FUNCTION_BLOCK _HRESULT_TestSuite EXTENDS TcUnit.FB_TestSuite
VAR
END_VAR

TestAddress();
TestClearReference();
TestClone();
TestTypeNameReturnsExpected();
TestIdentifierReturnsExpected();
TestMakeReferenceToFollowsReference();
TestMakeReferenceToUpdatesReference();
TestSize();
TestValueReturnsExpectedAfterInit();
TestValueReturnsExpectedAfterChange();
TestSerializeTypeWith();
TestSerializeWith();
TestTryDeserializeFrom();
TestTryMakeReferenceToFollowsReference();
TestTryMakeReferenceToUpdatesReference();

METHOD PUBLIC TestAddress
VAR
    _type : _HRESULT(S_OK);
    notExpected : PVOID := 0;
    actual : PVOID;
END_VAR
TEST('TestAddress');

actual := _type.Address;

AssertFalse(
    Condition := (notExpected = actual),
    Message := 'Type did not return a valid address.'
);

TEST_FINISHED();
END_METHOD

METHOD PUBLIC TestClearReference
VAR
    _type : _HRESULT(S_OK);
	target : HRESULT := S_OK;
    expected : HRESULT := S_OK;
    actual : HRESULT;
END_VAR
TEST('TestClearReference');

_type.MakeReferenceTo(target);
_type.ClearReference();
target := S_FALSE;

actual := _type.Value;

AssertEquals(
    Expected := expected,
    Actual := actual,
    Message := 'Value did not follow target change'
);

TEST_FINISHED();
END_METHOD

METHOD PUBLIC TestClone
VAR
    _type : _HRESULT(S_OK);
	clone : I_Datatype;
	isValidClone : BOOL;
	compareResult : DINT;
END_VAR
TEST('TestClone');

clone := _type.Clone();

isValidClone := clone <> 0;

IF isValidClone THEN
	compareResult := memcmp(_type.Address, clone.Address, clone.Size);
END_IF

AssertTrue(
	Condition := isValidClone,
	Message := 'Clone did not produce a clone'
);

AssertEquals_DINT(
	Expected := 0,
    Actual := compareResult,
    Message := 'Clone did not return a valid clone.'
);

clone.Dispose();

TEST_FINISHED();
END_METHOD

METHOD PUBLIC TestIdentifierReturnsExpected
VAR
    _type : _HRESULT(S_OK);
    expected : STRING := 'HRESULT';
    actual : STRING;
END_VAR
TEST('TestIdentifierReturnsExpected');

actual := _type.Identifier;

AssertEquals_STRING(
    Expected := expected,
    Actual := actual,
    Message := 'Type did not return correct iec type.'
);

TEST_FINISHED();
END_METHOD

METHOD PUBLIC TestMakeReferenceToFollowsReference
VAR
    _type : _HRESULT(S_OK);
	target : HRESULT := S_OK;
    expected : HRESULT := S_FALSE;
    actual : HRESULT;
END_VAR
TEST('TestMakeReferenceToFollowsReference');

_type.MakeReferenceTo(target);
target := S_FALSE;

actual := _type.Value;

AssertEquals(
    Expected := expected,
    Actual := actual,
    Message := 'Value did not follow target change'
);

TEST_FINISHED();
END_METHOD

METHOD PUBLIC TestMakeReferenceToUpdatesReference
VAR
    _type : _HRESULT(S_OK);
	target : HRESULT := S_OK;
    expected : HRESULT := S_FALSE;
    actual : HRESULT;
END_VAR
TEST('TestMakeReferenceToUpdatesReference');

_type.MakeReferenceTo(target);
_type.Value := S_FALSE;

actual := target;

AssertEquals(
    Expected := expected,
    Actual := actual,
    Message := 'Value did not update target'
);

TEST_FINISHED();
END_METHOD

METHOD PUBLIC TestSerializeTypeWith
VAR
    _type : _HRESULT(S_OK);
    serializer : JsonSerializer;
    expected : STRING(500) := '{"typeName":"ALIAS","identifier":"HRESULT","baseDatatype":{"typeName":"DINT","minValue":-2147483648,"maxValue":2147483647,"isSigned":true,"isFloat":false}}';
    actual : STRING(500);
END_VAR
TEST('TestSerializeTypeWith');

serializer.Reset();
_type.SerializeTypeWith(serializer);
serializer.TryGetSerializedData(ADR(actual), SIZEOF(actual));

AssertEquals_STRING(
    Expected := expected,
    Actual := actual,
    Message := 'Serialization of type did not return correct string.'
);

TEST_FINISHED();
END_METHOD

METHOD PUBLIC TestSerializeWith
VAR
    _type : _HRESULT(S_FALSE);
    serializer : JsonSerializer;
    expected : STRING := '1';
    actual : STRING(500);
END_VAR
TEST('TestSerializeWith');

serializer.Reset();
_type.SerializeWith(serializer);
serializer.TryGetSerializedData(ADR(actual), SIZEOF(actual));

AssertEquals_STRING(
    Expected := expected,
    Actual := actual,
    Message := 'Serialization of type data did not return correct string.'
);

TEST_FINISHED();
END_METHOD

METHOD PUBLIC TestSize
VAR
    _type : _HRESULT(S_OK);
    expected : UDINT := SIZEOF(HRESULT);
    actual : UDINT;
END_VAR
TEST('TestSize');

actual := _type.Size;

AssertEquals_UDINT(
    Expected := Expected,
    Actual := actual,
    Message := 'Type did not return the correct size.'
);

TEST_FINISHED();
END_METHOD

METHOD PUBLIC TestTryDeserializeFrom
VAR
    deserializer : JsonDeserializer;
    feedback : DeserializerFeedback;
    json : STRING := '0';
    _type : _HRESULT(S_OK);
    expected : HRESULT := S_OK;
    actual : HRESULT;
 END_VAR
TEST('TestTryDeserializeFrom');

deserializer.Reset();
deserializer.TryLoad(json);
_type.TryDeserializeFrom(Deserializer, Feedback);

actual := _type.Value;

AssertEquals(
    Expected := expected,
    Actual := actual,
    Message := 'Type did not deserialize correctly.'
);

TEST_FINISHED();
END_METHOD

METHOD PUBLIC TestTryMakeReferenceToFollowsReference
VAR
    _type : _HRESULT(S_OK);
	target : _HRESULT(S_OK);
    expected : HRESULT := S_FALSE;
    actual : HRESULT;
END_VAR
TEST('TestTryMakeReferenceToFollowsReference');

_type.TryMakeReferenceTo(target);
target.Value := S_FALSE;

actual := _type.Value;

AssertEquals(
    Expected := expected,
    Actual := actual,
    Message := 'Value did not follow target change'
);

TEST_FINISHED();
END_METHOD

METHOD PUBLIC TestTryMakeReferenceToUpdatesReference
VAR
    _type : _HRESULT(S_OK);
	target : _HRESULT(S_OK);
    expected : HRESULT := S_FALSE;
    actual : HRESULT;
END_VAR
TEST('TestTryMakeReferenceToUpdatesReference');

_type.TryMakeReferenceTo(target);
_type.Value := S_FALSE;

actual := target.Value;

AssertEquals(
    Expected := expected,
    Actual := actual,
    Message := 'Value did not update target'
);

TEST_FINISHED();
END_METHOD

METHOD PUBLIC TestTypeNameReturnsExpected
VAR
    _type : _HRESULT(S_OK);
    expected : STRING := 'ALIAS';
    actual : STRING;
END_VAR
TEST('TestTypeNameReturnsExpected');

actual := _type.TypeName;

AssertEquals_STRING(
    Expected := expected,
    Actual := actual,
    Message := 'Type did not return correct iec type.'
);

TEST_FINISHED();
END_METHOD

METHOD PUBLIC TestValueReturnsExpectedAfterChange
VAR
    _type : _HRESULT(S_OK);
    expected : HRESULT := S_FALSE;
    actual : HRESULT;
END_VAR
TEST('TestValueReturnsExpectedAfterChange');

_type.Value := S_FALSE;

actual := _type.Value;

AssertEquals(
    Expected := expected,
    Actual := actual,
    Message := 'Expected value not returned after change.'
);

TEST_FINISHED();
END_METHOD

METHOD PUBLIC TestValueReturnsExpectedAfterInit
VAR
    _type : _HRESULT(S_FALSE);
    expected : HRESULT := S_FALSE;
    actual : HRESULT;
END_VAR
TEST('TestValueReturnsExpectedAfterInit');

actual := _type.Value;

AssertEquals(
    Expected := expected,
    Actual := actual,
    Message := 'Expected value not returned after Init.'
);

TEST_FINISHED();
END_METHOD

END_FUNCTION_BLOCK

(* stored: Version 1.1.0.1, ProductVersion 3.1.4024.12
   POU _HRESULT_TestSuite: Id {3126607e-1658-0117-2d87-40eeac96a42f}, SpecialFunc None
   Method TestAddress: Id {f25dee84-18b5-0e37-372c-2dc32025c2b1}
   Method TestClearReference: Id {0dc2fdec-7c49-0140-0478-50a36a39a687}
   Method TestClone: Id {8f354877-490e-030c-0dba-9c34dc13f198}
   Method TestIdentifierReturnsExpected: Id {3165a4f6-4fed-0c9d-2598-66bcf8827de6}
   Method TestMakeReferenceToFollowsReference: Id {a76a35bb-e4a0-0fe6-3ede-dd228e426a2d}
   Method TestMakeReferenceToUpdatesReference: Id {c61f656f-b23b-0a46-2185-1bde701efbf7}
   Method TestSerializeTypeWith: Id {2500fb5f-6461-092c-1d90-89c01ddd73ad}
   Method TestSerializeWith: Id {106bab7d-0b4f-02de-137c-091f2f88c15a}
   Method TestSize: Id {4e5ac305-9227-0c2d-3b8d-c15d93c8d1eb}
   Method TestTryDeserializeFrom: Id {748ec791-ab28-04b2-3d9c-6c68cf44013f}
   Method TestTryMakeReferenceToFollowsReference: Id {eca1b1f7-8028-0c9d-1123-24e4860df742}
   Method TestTryMakeReferenceToUpdatesReference: Id {5be2926c-555a-0f58-2f90-e3e0c520061b}
   Method TestTypeNameReturnsExpected: Id {e4607604-b109-0a28-2dc4-95d9b03e4f5b}
   Method TestValueReturnsExpectedAfterChange: Id {55992bd8-f975-021f-35b7-039a0a9c4594}
   Method TestValueReturnsExpectedAfterInit: Id {86eacfa8-cb69-0c1d-3981-d4262702f0f3} *)
